FUNCTION_BLOCK FB_Message
VAR_INPUT
	eLogLevel:			E_LogLevel;
	nID:				UDINT;
	nTimestamp:			ULINT;	
	sSource:			STRING(255);
	sType:				STRING(255);
	sMessage:			STRING(255);
	sDefault:			STRING(255);
	sArguments:			STRING(255);
	bRaised:			BOOL;
END_VAR
VAR_OUTPUT
END_VAR
VAR
END_VAR

END_FUNCTION_BLOCK

(* stored: Version 1.1.0.1
   POU FB_Message: Id {84167246-7318-466e-9219-bf236e6d60e2}, SpecialFunc None *)
